INTERFACE I_DriveCmd

PROPERTY CommandedAborted : BOOL
GET
END_GET
END_PROPERTY

PROPERTY CommandHalt : BOOL
GET
END_GET
SET
END_SET
END_PROPERTY

PROPERTY CommandMoveAbsolute : BOOL
GET
END_GET
SET
END_SET
END_PROPERTY

PROPERTY CommandMoveHome : BOOL
GET
END_GET
SET
END_SET
END_PROPERTY

PROPERTY CommandReset : BOOL
GET
END_GET
SET
END_SET
END_PROPERTY

METHOD ErrorHandling
VAR_INPUT
END_VAR
END_METHOD

(*
    Check all post condition before updating bCommandedMoveAbsolute
    The implmentatation will depend on the axis type
    DS402 NC/Direct axis : Implementation need to check that the drive is in the correct mode before initaiting the move then set bCommandedMoveAbsolute
    MP NC axis : will immediately write to bCommandedMoveAbsolute
*)
METHOD StartMove : BOOL
VAR_INPUT
	MoveMode	: E_EpicsMotorCmd;
	CmdExecute	: BOOL;
END_VAR
END_METHOD

END_INTERFACE

(* stored: Version 1.1.0.1
   Itf I_DriveCmd: Id {32204644-5c98-476b-85f8-dcfa96ca1a0e}
   Property CommandedAborted: Id {1d99348a-3430-4255-9b3c-9dce426a062e}
   Get Get: Id {cbcc2716-a4d8-4b53-a6de-05baab07ff72}
   Property CommandHalt: Id {28caa621-b1b5-45c3-948b-355529ae63c2}
   Get Get: Id {9fc451d3-9985-4a65-a079-615be98f9e47}
   Set Set: Id {afbd26a2-5d4f-4673-a5ff-92792f920642}
   Property CommandMoveAbsolute: Id {be1022ab-c175-45cf-b747-4904f7dbb61a}
   Get Get: Id {2b465d88-c80e-452d-bd64-a4daa37a937f}
   Set Set: Id {148eb03e-69c6-4884-b363-b91c6e29515e}
   Property CommandMoveHome: Id {c447ca24-e237-4885-a9a3-281864c8338b}
   Get Get: Id {bd009231-61d7-4bed-ae68-5c589c9f60c3}
   Set Set: Id {fd07a648-391b-4835-a127-b5f46d9080b8}
   Property CommandReset: Id {cd7e8bfd-a0cf-4671-a69b-1557a160bd00}
   Get Get: Id {cc6afb54-414e-4354-b571-2acc42bfca27}
   Set Set: Id {367e203b-5f9b-41d7-9061-a806fa5317d7}
   Method ErrorHandling: Id {8c3f2673-8367-4245-8039-269c7637bb4c}
   Method StartMove: Id {2d898c45-221d-4ab1-9add-83136ca35be3} *)
